(* IEC 61131-3 sources: RL_MAR/experiments/comparison/llm4plc/results/deepseek-ai-DeepSeek-V3.2_20260506_104945/20260506_114714, 4 files *)

(* ---- generated_code_iteration_0.st ---- *)
START_ST
FUNCTION_BLOCK RetractableRoofControl
VAR_INPUT
    RainSensor : BOOL; (* Input to detect rain *)
    WindSensor : BOOL; (* Input to detect wind *)
    TemperatureSensor : REAL; (* Input to measure temperature *)
END_VAR
VAR_OUTPUT
    RoofMotor : BOOL; (* Output to control the roof motor *)
END_VAR
VAR
    state : INT; (* The current state variable *)
    prevState : INT; (* The previous state variable (optional, for debugging or transition logging) *)
END_VAR

(* State definitions *)
CONST
    STATE_IDLE : INT := 0;
    STATE_CLOSE_COMPLETELY : INT := 1;
    STATE_PARTIALLY_CLOSE : INT := 2;
    STATE_CLOSE_SLIGHTLY : INT := 3;
    STATE_FULLY_OPEN : INT := 4;
END_CONST

(* Main state machine logic *)
CASE state OF
    STATE_IDLE:
        (* Output for STATE_IDLE: RoofMotor = FALSE (or maintain previous state, but typically OFF for initialization) *)
        RoofMotor := FALSE;

        (* Transitions from STATE_IDLE *)
        IF RainSensor AND WindSensor THEN
            state := STATE_CLOSE_COMPLETELY;
        ELSIF RainSensor AND NOT WindSensor THEN
            state := STATE_PARTIALLY_CLOSE;
        ELSIF NOT RainSensor AND TemperatureSensor < 20.0 THEN
            state := STATE_CLOSE_SLIGHTLY;
        ELSIF NOT RainSensor AND TemperatureSensor >= 20.0 THEN
            state := STATE_FULLY_OPEN;
        END_IF;

    STATE_CLOSE_COMPLETELY:
        (* Output for STATE_CLOSE_COMPLETELY: RoofMotor = FALSE (Motor OFF to close completely) *)
        RoofMotor := FALSE;

        (* Transitions from STATE_CLOSE_COMPLETELY *)
        IF RainSensor AND NOT WindSensor THEN
            state := STATE_PARTIALLY_CLOSE;
        ELSIF NOT RainSensor AND TemperatureSensor < 20.0 THEN
            state := STATE_CLOSE_SLIGHTLY;
        ELSIF NOT RainSensor AND TemperatureSensor >= 20.0 THEN
            state := STATE_FULLY_OPEN;
        END_IF;

    STATE_PARTIALLY_CLOSE:
        (* Output for STATE_PARTIALLY_CLOSE: RoofMotor = TRUE (Motor ON to partially close) *)
        RoofMotor := TRUE;

        (* Transitions from STATE_PARTIALLY_CLOSE *)
        IF RainSensor AND WindSensor THEN
            state := STATE_CLOSE_COMPLETELY;
        ELSIF NOT RainSensor AND TemperatureSensor < 20.0 THEN
            state := STATE_CLOSE_SLIGHTLY;
        ELSIF NOT RainSensor AND TemperatureSensor >= 20.0 THEN
            state := STATE_FULLY_OPEN;
        END_IF;

    STATE_CLOSE_SLIGHTLY:
        (* Output for STATE_CLOSE_SLIGHTLY: RoofMotor = TRUE (Motor ON to close slightly) *)
        RoofMotor := TRUE;

        (* Transitions from STATE_CLOSE_SLIGHTLY *)
        IF RainSensor AND WindSensor THEN
            state := STATE_CLOSE_COMPLETELY;
        ELSIF RainSensor AND NOT WindSensor THEN
            state := STATE_PARTIALLY_CLOSE;
        ELSIF NOT RainSensor AND TemperatureSensor >= 20.0 THEN
            state := STATE_FULLY_OPEN;
        END_IF;

    STATE_FULLY_OPEN:
        (* Output for STATE_FULLY_OPEN: RoofMotor = FALSE (Motor OFF to be fully open) *)
        RoofMotor := FALSE;

        (* Transitions from STATE_FULLY_OPEN *)
        IF RainSensor AND WindSensor THEN
            state := STATE_CLOSE_COMPLETELY;
        ELSIF RainSensor AND NOT WindSensor THEN
            state := STATE_PARTIALLY_CLOSE;
        ELSIF NOT RainSensor AND TemperatureSensor < 20.0 THEN
            state := STATE_CLOSE_SLIGHTLY;
        END_IF;

    ELSE
        (* Default case: reset to IDLE state *)
        state := STATE_IDLE;
        RoofMotor := FALSE;
END_CASE;

(* Optional: Store previous state for debugging or logging *)
prevState := state;

END_FUNCTION_BLOCK
END_ST

(* ---- generated_code_iteration_1.st ---- *)
START_REASON
The validation feedback indicates a CODESYS compiler error: "应该用';' 替换'STATE_IDLE'". This is a Chinese error message meaning "should replace 'STATE_IDLE' with ';'". This suggests a syntax issue with the CONST declaration. In CODESYS Structured Text, CONST sections must end with a semicolon (;) after each constant declaration, not a comma. Looking at the original code:

CONST
    STATE_IDLE : INT := 0;
    STATE_CLOSE_COMPLETELY : INT := 1;
    STATE_PARTIALLY_CLOSE : INT := 2;
    STATE_CLOSE_SLIGHTLY : INT := 3;
    STATE_FULLY_OPEN : INT := 4;
END_CONST

The syntax appears correct with semicolons. However, the error message specifically mentions 'STATE_IDLE', which might indicate that the compiler is interpreting something incorrectly. Possibly the issue is that the CONST section is placed inside the FUNCTION_BLOCK but not properly within a VAR_CONSTANT section. In CODESYS, constants should be declared in a VAR_CONSTANT block, not with CONST/END_CONST. The correct syntax is:

VAR_CONSTANT
    STATE_IDLE : INT := 0;
    STATE_CLOSE_COMPLETELY : INT := 1;
    STATE_PARTIALLY_CLOSE : INT := 2;
    STATE_CLOSE_SLIGHTLY : INT := 3;
    STATE_FULLY_OPEN : INT := 4;
END_VAR

Alternatively, if using global constants, they should be defined outside the FUNCTION_BLOCK. But since this is a FUNCTION_BLOCK, internal constants should use VAR_CONSTANT. The original code used CONST/END_CONST, which might not be valid in CODESYS ST. I will change this to VAR_CONSTANT to fix the compiler error.
END_REASON

START_ST
FUNCTION_BLOCK RetractableRoofControl
VAR_INPUT
    RainSensor : BOOL; (* Input to detect rain *)
    WindSensor : BOOL; (* Input to detect wind *)
    TemperatureSensor : REAL; (* Input to measure temperature *)
END_VAR
VAR_OUTPUT
    RoofMotor : BOOL; (* Output to control the roof motor *)
END_VAR
VAR
    state : INT; (* The current state variable *)
    prevState : INT; (* The previous state variable (optional, for debugging or transition logging) *)
END_VAR
VAR_CONSTANT
    STATE_IDLE : INT := 0;
    STATE_CLOSE_COMPLETELY : INT := 1;
    STATE_PARTIALLY_CLOSE : INT := 2;
    STATE_CLOSE_SLIGHTLY : INT := 3;
    STATE_FULLY_OPEN : INT := 4;
END_VAR

(* Main state machine logic *)
CASE state OF
    STATE_IDLE:
        (* Output for STATE_IDLE: RoofMotor = FALSE (or maintain previous state, but typically OFF for initialization) *)
        RoofMotor := FALSE;

        (* Transitions from STATE_IDLE *)
        IF RainSensor AND WindSensor THEN
            state := STATE_CLOSE_COMPLETELY;
        ELSIF RainSensor AND NOT WindSensor THEN
            state := STATE_PARTIALLY_CLOSE;
        ELSIF NOT RainSensor AND TemperatureSensor < 20.0 THEN
            state := STATE_CLOSE_SLIGHTLY;
        ELSIF NOT RainSensor AND TemperatureSensor >= 20.0 THEN
            state := STATE_FULLY_OPEN;
        END_IF;

    STATE_CLOSE_COMPLETELY:
        (* Output for STATE_CLOSE_COMPLETELY: RoofMotor = FALSE (Motor OFF to close completely) *)
        RoofMotor := FALSE;

        (* Transitions from STATE_CLOSE_COMPLETELY *)
        IF RainSensor AND NOT WindSensor THEN
            state := STATE_PARTIALLY_CLOSE;
        ELSIF NOT RainSensor AND TemperatureSensor < 20.0 THEN
            state := STATE_CLOSE_SLIGHTLY;
        ELSIF NOT RainSensor AND TemperatureSensor >= 20.0 THEN
            state := STATE_FULLY_OPEN;
        END_IF;

    STATE_PARTIALLY_CLOSE:
        (* Output for STATE_PARTIALLY_CLOSE: RoofMotor = TRUE (Motor ON to partially close) *)
        RoofMotor := TRUE;

        (* Transitions from STATE_PARTIALLY_CLOSE *)
        IF RainSensor AND WindSensor THEN
            state := STATE_CLOSE_COMPLETELY;
        ELSIF NOT RainSensor AND TemperatureSensor < 20.0 THEN
            state := STATE_CLOSE_SLIGHTLY;
        ELSIF NOT RainSensor AND TemperatureSensor >= 20.0 THEN
            state := STATE_FULLY_OPEN;
        END_IF;

    STATE_CLOSE_SLIGHTLY:
        (* Output for STATE_CLOSE_SLIGHTLY: RoofMotor = TRUE (Motor ON to close slightly) *)
        RoofMotor := TRUE;

        (* Transitions from STATE_CLOSE_SLIGHTLY *)
        IF RainSensor AND WindSensor THEN
            state := STATE_CLOSE_COMPLETELY;
        ELSIF RainSensor AND NOT WindSensor THEN
            state := STATE_PARTIALLY_CLOSE;
        ELSIF NOT RainSensor AND TemperatureSensor >= 20.0 THEN
            state := STATE_FULLY_OPEN;
        END_IF;

    STATE_FULLY_OPEN:
        (* Output for STATE_FULLY_OPEN: RoofMotor = FALSE (Motor OFF to be fully open) *)
        RoofMotor := FALSE;

        (* Transitions from STATE_FULLY_OPEN *)
        IF RainSensor AND WindSensor THEN
            state := STATE_CLOSE_COMPLETELY;
        ELSIF RainSensor AND NOT WindSensor THEN
            state := STATE_PARTIALLY_CLOSE;
        ELSIF NOT RainSensor AND TemperatureSensor < 20.0 THEN
            state := STATE_CLOSE_SLIGHTLY;
        END_IF;

    ELSE
        (* Default case: reset to IDLE state *)
        state := STATE_IDLE;
        RoofMotor := FALSE;
END_CASE;

(* Optional: Store previous state for debugging or logging *)
prevState := state;

END_FUNCTION_BLOCK
END_ST

(* ---- generated_code_iteration_2.st ---- *)
START_REASON
The validation feedback indicates an encoding issue: "ANTLR syntax check failed: 'gbk' codec can't decode byte 0xaf in position 79: illegal multibyte sequence". This error occurs because the compiler (likely using GBK encoding for Chinese systems) encounters a non-GBK character in the code, specifically at position 79. This is often due to special characters like curly quotes, em dashes, or non-ASCII characters in comments. Looking at the previous code, the comments contain standard ASCII characters, but there might be an invisible or special character introduced. The position 79 suggests it's early in the code, possibly in the FUNCTION_BLOCK declaration or first comments. To fix this, I need to ensure all characters are ASCII-compatible. I will rewrite the code using only ASCII characters in comments and remove any potential non-ASCII characters. I'll also simplify comments to avoid any special formatting.
END_REASON

START_ST
FUNCTION_BLOCK RetractableRoofControl
VAR_INPUT
    RainSensor : BOOL;
    WindSensor : BOOL;
    TemperatureSensor : REAL;
END_VAR
VAR_OUTPUT
    RoofMotor : BOOL;
END_VAR
VAR
    state : INT;
    prevState : INT;
END_VAR
VAR_CONSTANT
    STATE_IDLE : INT := 0;
    STATE_CLOSE_COMPLETELY : INT := 1;
    STATE_PARTIALLY_CLOSE : INT := 2;
    STATE_CLOSE_SLIGHTLY : INT := 3;
    STATE_FULLY_OPEN : INT := 4;
END_VAR

CASE state OF
    STATE_IDLE:
        RoofMotor := FALSE;
        IF RainSensor AND WindSensor THEN
            state := STATE_CLOSE_COMPLETELY;
        ELSIF RainSensor AND NOT WindSensor THEN
            state := STATE_PARTIALLY_CLOSE;
        ELSIF NOT RainSensor AND TemperatureSensor < 20.0 THEN
            state := STATE_CLOSE_SLIGHTLY;
        ELSIF NOT RainSensor AND TemperatureSensor >= 20.0 THEN
            state := STATE_FULLY_OPEN;
        END_IF;

    STATE_CLOSE_COMPLETELY:
        RoofMotor := FALSE;
        IF RainSensor AND NOT WindSensor THEN
            state := STATE_PARTIALLY_CLOSE;
        ELSIF NOT RainSensor AND TemperatureSensor < 20.0 THEN
            state := STATE_CLOSE_SLIGHTLY;
        ELSIF NOT RainSensor AND TemperatureSensor >= 20.0 THEN
            state := STATE_FULLY_OPEN;
        END_IF;

    STATE_PARTIALLY_CLOSE:
        RoofMotor := TRUE;
        IF RainSensor AND WindSensor THEN
            state := STATE_CLOSE_COMPLETELY;
        ELSIF NOT RainSensor AND TemperatureSensor < 20.0 THEN
            state := STATE_CLOSE_SLIGHTLY;
        ELSIF NOT RainSensor AND TemperatureSensor >= 20.0 THEN
            state := STATE_FULLY_OPEN;
        END_IF;

    STATE_CLOSE_SLIGHTLY:
        RoofMotor := TRUE;
        IF RainSensor AND WindSensor THEN
            state := STATE_CLOSE_COMPLETELY;
        ELSIF RainSensor AND NOT WindSensor THEN
            state := STATE_PARTIALLY_CLOSE;
        ELSIF NOT RainSensor AND TemperatureSensor >= 20.0 THEN
            state := STATE_FULLY_OPEN;
        END_IF;

    STATE_FULLY_OPEN:
        RoofMotor := FALSE;
        IF RainSensor AND WindSensor THEN
            state := STATE_CLOSE_COMPLETELY;
        ELSIF RainSensor AND NOT WindSensor THEN
            state := STATE_PARTIALLY_CLOSE;
        ELSIF NOT RainSensor AND TemperatureSensor < 20.0 THEN
            state := STATE_CLOSE_SLIGHTLY;
        END_IF;

    ELSE
        state := STATE_IDLE;
        RoofMotor := FALSE;
END_CASE;

prevState := state;

END_FUNCTION_BLOCK
END_ST

(* ---- generated_code_iteration_3.st ---- *)
START_REASON
The validation feedback indicates that the CODESYS compiler validation failed because of the use of "VAR_CONSTANT". The feedback states: "应该采用VAR, VAR_INPUT, VAR_OUTPUT 或 VAR_IN_OUT 取代VAR_CONSTANT". This means that in CODESYS Structured Text, "VAR_CONSTANT" is not a valid keyword for declaring constants inside a FUNCTION_BLOCK. Instead, constants should be declared within the VAR section using the "CONSTANT" attribute. I need to replace the VAR_CONSTANT section with a VAR section where the constants are declared with the "CONSTANT" keyword. This is a common syntax difference between CODESYS and other PLC programming environments. I will adjust the code accordingly to comply with CODESYS standards.
END_REASON

START_ST
FUNCTION_BLOCK RetractableRoofControl
VAR_INPUT
    RainSensor : BOOL;
    WindSensor : BOOL;
    TemperatureSensor : REAL;
END_VAR
VAR_OUTPUT
    RoofMotor : BOOL;
END_VAR
VAR
    state : INT;
    prevState : INT;
END_VAR
VAR
    STATE_IDLE : INT := 0;
    STATE_CLOSE_COMPLETELY : INT := 1;
    STATE_PARTIALLY_CLOSE : INT := 2;
    STATE_CLOSE_SLIGHTLY : INT := 3;
    STATE_FULLY_OPEN : INT := 4;
END_VAR

CASE state OF
    STATE_IDLE:
        RoofMotor := FALSE;
        IF RainSensor AND WindSensor THEN
            state := STATE_CLOSE_COMPLETELY;
        ELSIF RainSensor AND NOT WindSensor THEN
            state := STATE_PARTIALLY_CLOSE;
        ELSIF NOT RainSensor AND TemperatureSensor < 20.0 THEN
            state := STATE_CLOSE_SLIGHTLY;
        ELSIF NOT RainSensor AND TemperatureSensor >= 20.0 THEN
            state := STATE_FULLY_OPEN;
        END_IF;

    STATE_CLOSE_COMPLETELY:
        RoofMotor := FALSE;
        IF RainSensor AND NOT WindSensor THEN
            state := STATE_PARTIALLY_CLOSE;
        ELSIF NOT RainSensor AND TemperatureSensor < 20.0 THEN
            state := STATE_CLOSE_SLIGHTLY;
        ELSIF NOT RainSensor AND TemperatureSensor >= 20.0 THEN
            state := STATE_FULLY_OPEN;
        END_IF;

    STATE_PARTIALLY_CLOSE:
        RoofMotor := TRUE;
        IF RainSensor AND WindSensor THEN
            state := STATE_CLOSE_COMPLETELY;
        ELSIF NOT RainSensor AND TemperatureSensor < 20.0 THEN
            state := STATE_CLOSE_SLIGHTLY;
        ELSIF NOT RainSensor AND TemperatureSensor >= 20.0 THEN
            state := STATE_FULLY_OPEN;
        END_IF;

    STATE_CLOSE_SLIGHTLY:
        RoofMotor := TRUE;
        IF RainSensor AND WindSensor THEN
            state := STATE_CLOSE_COMPLETELY;
        ELSIF RainSensor AND NOT WindSensor THEN
            state := STATE_PARTIALLY_CLOSE;
        ELSIF NOT RainSensor AND TemperatureSensor >= 20.0 THEN
            state := STATE_FULLY_OPEN;
        END_IF;

    STATE_FULLY_OPEN:
        RoofMotor := FALSE;
        IF RainSensor AND WindSensor THEN
            state := STATE_CLOSE_COMPLETELY;
        ELSIF RainSensor AND NOT WindSensor THEN
            state := STATE_PARTIALLY_CLOSE;
        ELSIF NOT RainSensor AND TemperatureSensor < 20.0 THEN
            state := STATE_CLOSE_SLIGHTLY;
        END_IF;

    ELSE
        state := STATE_IDLE;
        RoofMotor := FALSE;
END_CASE;

prevState := state;

END_FUNCTION_BLOCK
END_ST
